// TIA Portal V20 program export: 1 tag tables, 3 data types, 0 data blocks, 4 code blocks (in call order from the OBs), 0 instance data blocks

VAR_GLOBAL   // PLC tag table "TagTable_AI"
   AHU1_RAT_Temp AT  : Real;
   AHU1_OAT_Temp AT  : Real;
   AHU1_DAT_Temp AT  : Real;
   AHU1_CW_VlvFdbk AT  : Real;
   AHU1_HW_VlvFdbk AT  : Real;
   AHU1_DMP_PosFdbk AT  : Real;
END_VAR

TYPE "UDT200_EM_Cooling"
   STRUCT
      CHW_Freeze_Stat_DI : Bool;   // Digital Input: Freeze-stat on chilled water coil (`True` = Fault).
      CHW_Valve_Fdbk_AI : Real;   // Analog Input: Chilled water valve position feedback (0-100%).
      CHW_Valve_Cmd_AO : Real;   // Analog Output: Chilled water valve position command (0-100%).
      CHW_Freeze_Alm : Bool;   // Alarm: Chilled water coil freeze-stat has tripped.
      Valve_Failure_Alm : Bool;   // Alarm: `True` if valve command and feedback do not match.
   END_STRUCT;
END_TYPE

TYPE "UDT300_EM_Heating"
   STRUCT
      HW_Freeze_Stat_DI : Bool;   // Digital Input: Freeze-stat on hot water coil (`True` = Fault).
      HW_Valve_Fdbk_AI : Real;   // Analog Input: Hot water valve position feedback (0-100%).
      HW_Valve_Cmd_AO : Real;   // Analog Output: Hot water valve position command (0-100%).
      HW_Freeze_Alm : Bool;   // Alarm: Hot water coil freeze-stat has tripped.
      Valve_Failure_Alm : Bool;   // Alarm: `True` if valve command and feedback do not match.
   END_STRUCT;
END_TYPE

TYPE "UDT400_EM_Damper"
   STRUCT
      Return_Air_Temp_AI : Real;   // Analog Input: Return air temperature sensor.
      Outside_Air_Temp_AI : Real;   // Analog Input: Outside air temperature sensor.
      Discharge_Air_Temp_AI : Real;   // Analog Input: Discharge air temperature sensor.
      Damper_Pos_Fdbk_AI : Real;   // Analog Input: Damper position feedback (0-100%).
      Damper_Pos_Cmd_AO : Real;   // Analog Output: Damper position command (0.0 - 100.0 %).
      Damper_Failure_Alm : Bool;   // Alarm: `True` if damper command and feedback do not match.
      Min_Fresh_Air_Pos : Real;   // Minimum damper position for ventilation (e.g., 20.0 %).
      Econ_Temp_Diff : Real;   // Temp diff (RAT - OAT) to enable economizer (e.g., 2.0).
      Econ_High_Limit : Real;   // High OAT limit to disable economizer (e.g., 65.0).
      Econ_Mode_Active : Bool;   // Status: `True` when economizer mode is active.
   END_STRUCT;
END_TYPE

ORGANIZATION_BLOCK "OB1_Main"   // OB1, SCL
TITLE = Main Program [OB1]
AUTHOR : Jules
VERSION : 0.1
// Main program block for the AHU Controller. Contains all I/O mapping, control logic, and FB calls.
// stored: AutoNumber false, IsOptimized true
BEGIN
   REGION INPUT MAPPING 
   (/**/) "IDB_SupplyFan".UDT.Run_Fdbk_DI := "AHU1_SF_RunFdbk";
   "IDB_SupplyFan".UDT.Airflow_Status_DI := "AHU1_SF_AirflowSw";
   "IDB_SupplyFan".UDT.VFD_Fault_DI := "AHU1_SF_VfdFault";
   "IDB_Cooling".UDT.CHW_Freeze_Stat_DI := "AHU1_CW_FreezeStat";
   "IDB_Cooling".UDT.CHW_Valve_Fdbk_AI := "AHU1_CW_VlvFdbk";
   "IDB_Heating".UDT.HW_Freeze_Stat_DI := "AHU1_HW_FreezeStat";
   "IDB_Heating".UDT.HW_Valve_Fdbk_AI := "AHU1_HW_VlvFdbk";
   "IDB_Damper".UDT.Return_Air_Temp_AI := "AHU1_RAT_Temp";
   "IDB_Damper".UDT.Outside_Air_Temp_AI := "AHU1_OAT_Temp";
   "IDB_Damper".UDT.Discharge_Air_Temp_AI := "AHU1_DAT_Temp";
   "IDB_Damper".UDT.Damper_Pos_Fdbk_AI := "AHU1_DMP_PosFdbk";
   "IDB_Monitoring".UDT.Dirty_Filter_DI := "AHU1_SYS_DirtyFilter";
   END_REGION

   REGION MAIN CONTROL LOGIC 
   (/**/) (/**/) (/**/) (/**/) (/**/) (/**/) (/**/) (/**/) (/**/) (/**/) (/**/) (/**/) (/**/) (/**/)END_REGION

   REGION FUNCTION BLOCK CALLS 
   (/**/) "IDB_SupplyFan"(Enable:= TRUE);(/**/) "IDB_Cooling"(Enable:= TRUE, Valve_Demand_In:= 0.0);(/**/) "IDB_Heating"(Enable:= TRUE, Valve_Demand_In:= 0.0);(/**/) "IDB_Damper"(Enable:= TRUE);
   "IDB_Monitoring"(Enable:= TRUE);
   END_REGION

   REGION OUTPUT MAPPING 
   (/**/) "AHU1_SF_StartCmd" := "IDB_SupplyFan".UDT.Start_Cmd_DO;
   "AHU1_SF_SpeedRef" := "IDB_SupplyFan".UDT.Speed_Ref_AO;
   "AHU1_CW_VlvCmd" := "IDB_Cooling".UDT.CHW_Valve_Cmd_AO;
   "AHU1_HW_VlvCmd" := "IDB_Heating".UDT.HW_Valve_Cmd_AO;
   "AHU1_DMP_PosCmd" := "IDB_Damper".UDT.Damper_Pos_Cmd_AO;
   END_REGION
END_ORGANIZATION_BLOCK

FUNCTION_BLOCK "FB200_EM_Cooling"   // FB, SCL
TITLE = EM-200: Cooling Control
AUTHOR : Dallas Levine
VERSION : 0.1
// This block contains all logic for the Cooling Equipment Module (EM-200).
// stored: AutoNumber true, IsRetain false
   VAR_INPUT
      Enable : Bool;   // Enables the block's execution.
      Valve_Demand_In : Real;   // Demand signal from the main PID controller (0.0 - 100.0 %).
   END_VAR
   VAR
      UDT : "UDT200_EM_Cooling";   // The data interface for the Cooling Equipment Module.
      Feedback_Fault_Timer : TON_TIME;   // Timer for the feedback fault delay.
   END_VAR
   VAR CONSTANT
      FEEDBACK_TOLERANCE : Real := 10.0;   // Allowable deviation between command and feedback (%).
      FEEDBACK_DELAY : Time := T#60s;   // Time delay before a feedback mismatch becomes an alarm.
   END_VAR
BEGIN
   REGION Main Logic 
   IF #Enable THEN

    (/**/) #UDT.CHW_Valve_Cmd_AO := #Valve_Demand_In;

    (/**/) #UDT.CHW_Freeze_Alm := #UDT.CHW_Freeze_Stat_DI;
    IF #UDT.CHW_Freeze_Alm THEN
     #UDT.CHW_Valve_Cmd_AO := 0.0;
    END_IF;

    (/**/) #Feedback_Fault_Timer(IN:= ABS(FV:=#UDT.CHW_Valve_Cmd_AO - #UDT.CHW_Valve_Fdbk_AI) > #FEEDBACK_TOLERANCE,
           PT:= #FEEDBACK_DELAY);
    #UDT.Valve_Failure_Alm := #Feedback_Fault_Timer.Q;
   ELSE
    (/**/) #UDT.CHW_Valve_Cmd_AO := 0.0;
    #UDT.Valve_Failure_Alm := FALSE;
   END_IF;
   END_REGION
END_FUNCTION_BLOCK

FUNCTION_BLOCK "FB300_EM_Heating"   // FB, SCL
TITLE = EM-300: Heating Control
AUTHOR : Dallas Levine
VERSION : 0.1
// This block contains all logic for the Heating Equipment Module (EM-300).
// stored: AutoNumber true, IsRetain false
   VAR_INPUT
      Enable : Bool;   // Enables the block's execution.
      Valve_Demand_In : Real;   // Demand signal from the main PID controller (0.0 - 100.0 %).
   END_VAR
   VAR
      UDT : "UDT300_EM_Heating";   // The data interface for the Heating Equipment Module.
      Feedback_Fault_Timer : TON_TIME;   // Timer for the feedback fault delay.
   END_VAR
   VAR CONSTANT
      FEEDBACK_TOLERANCE : Real := 10.0;   // Allowable deviation between command and feedback (%).
      FEEDBACK_DELAY : Time := T#60s;   // Time delay before a feedback mismatch becomes an alarm.
   END_VAR
BEGIN
   REGION Main Logic 
   IF #Enable THEN

    (/**/) #UDT.HW_Valve_Cmd_AO := #Valve_Demand_In;

    (/**/) #UDT.HW_Freeze_Alm := #UDT.HW_Freeze_Stat_DI;
    IF #UDT.HW_Freeze_Alm THEN
     #UDT.HW_Valve_Cmd_AO := 0.0;
    END_IF;

    (/**/) #Feedback_Fault_Timer(IN:= ABS(FV:=#UDT.HW_Valve_Cmd_AO - #UDT.HW_Valve_Fdbk_AI) > #FEEDBACK_TOLERANCE,
           PT:= #FEEDBACK_DELAY);
    #UDT.Valve_Failure_Alm := #Feedback_Fault_Timer.Q;
   ELSE
    (/**/) #UDT.HW_Valve_Cmd_AO := 0.0;
    #UDT.Valve_Failure_Alm := FALSE;
   END_IF;
   END_REGION
END_FUNCTION_BLOCK

FUNCTION_BLOCK "FB400_EM_Damper"   // FB, SCL
TITLE = EM-400: Damper Control
AUTHOR : Dallas Levine
VERSION : 0.1
// This block contains all logic for the Damper Equipment Module (EM-400).
// stored: AutoNumber true, IsRetain false
   VAR_INPUT
      Enable : Bool;   // Enables the block's execution.
   END_VAR
   VAR
      UDT : "UDT400_EM_Damper";   // The data interface for the Damper Equipment Module.
      Feedback_Fault_Timer : TON_TIME;   // Timer for the feedback fault delay.
   END_VAR
   VAR CONSTANT
      FEEDBACK_TOLERANCE : Real := 10.0;   // Allowable deviation between command and feedback (%).
      FEEDBACK_DELAY : Time := T#60s;   // Time delay before a feedback mismatch becomes an alarm.
   END_VAR
BEGIN
   REGION Main Logic 
   IF #Enable THEN
    (/**/) #Feedback_Fault_Timer(IN:= ABS(FV:=#UDT.Damper_Pos_Cmd_AO - #UDT.Damper_Pos_Fdbk_AI) > #FEEDBACK_TOLERANCE,
           PT:= #FEEDBACK_DELAY);
    #UDT.Damper_Failure_Alm := #Feedback_Fault_Timer.Q;
   ELSE
    (/**/) #UDT.Damper_Failure_Alm := FALSE;
   END_IF;
   END_REGION
END_FUNCTION_BLOCK
